Staubli VAL3: getTool.pgx

public program getTool(num& x_nTool (dimensions=1))
begin
  // edit one
  x_nTool=pEditPoint.nIndexTool
end
